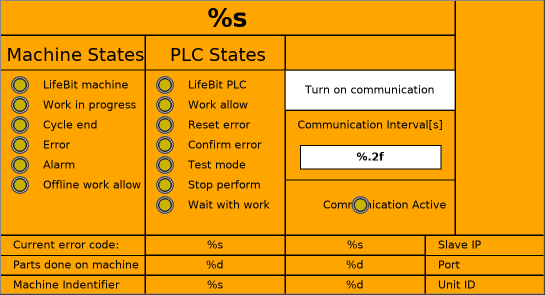
VISUALIZATION vChiniseMachineStatus_v2  // 545x295
VAR_IN_OUT
	stData					:	stChiniseMachineHmiData;
	stParams				:	stModTcpSlaveParams;
END_VAR
    Rectangle (285,35 170x200)
    Rectangle (0,235 145x60)
    Rectangle (0,35 145x200)
    Rectangle (0,35 455x35)
    Rectangle (145,35 140x200)
    Lamp1 (10,75 20x20), variable: stData.stPimCommunicationData.bLifeBitMachine, style: Lamp-Lamp1-Yellow
    Label (40,75 150x20), "LifeBit machine"
    Label (5,40 141x30), "Machine States"
    Lamp1 (10,95 20x20), variable: stData.stPimCommunicationData.bWorkInProgress, style: Lamp-Lamp1-Yellow
    Label (40,95 150x20), "Work in progress"
    Lamp1 (10,115 20x20), variable: stData.stPimCommunicationData.bCycleEnd, style: Lamp-Lamp1-Yellow
    Label (40,115 150x20), "Cycle end"
    Lamp1 (10,135 20x20), variable: stData.stPimCommunicationData.bError, style: Lamp-Lamp1-Yellow
    Label (40,135 150x20), "Error"
    Lamp1 (10,155 20x20), variable: stData.stPimCommunicationData.bAlarm, style: Lamp-Lamp1-Yellow
    Label (40,155 150x20), "Alarm"
    Lamp1 (10,175 20x20), variable: stData.stPimCommunicationData.bOfflineWorkAllow, style: Lamp-Lamp1-Yellow
    Label (40,175 150x20), "Offline work allow"
    Lamp1 (155,75 20x20), variable: stData.stPimCommunicationData.bLifeBitPLC, style: Lamp-Lamp1-Yellow
    Label (185,75 150x20), "LifeBit PLC"
    Label (150,40 136x30), "PLC States"
    Lamp1 (155,95 20x20), variable: stData.stPimCommunicationData.bWorkAllow, style: Lamp-Lamp1-Yellow
    Label (185,95 150x20), "Work allow"
    Lamp1 (155,115 20x20), variable: stData.stPimCommunicationData.bResetError, style: Lamp-Lamp1-Yellow
    Label (185,115 150x20), "Reset error"
    Lamp1 (155,135 20x20), variable: stData.stPimCommunicationData.bConfirmError, style: Lamp-Lamp1-Yellow
    Label (185,135 150x20), "Confirm error"
    Lamp1 (155,155 20x20), variable: stData.stPimCommunicationData.bTestMode, style: Lamp-Lamp1-Yellow
    Label (185,155 150x20), "Test mode"
    Lamp1 (155,175 20x20), variable: stData.stPimCommunicationData.bStopPerform, style: Lamp-Lamp1-Yellow
    Label (185,175 150x20), "Stop perform"
    Lamp1 (155,195 20x20), variable: stData.stPimCommunicationData.bWaitWithWork, style: Lamp-Lamp1-Yellow
    Label (185,195 150x20), "Wait with work"
    Rectangle (145,235 140x20), "%s", text variable: stData.stPimCommunicationData.iErrorCode
    Label (10,235 150x20), "Current error code:"
    Rectangle (0,0 455x35), "%s", text variable: stData.stModbusTcpData.sMachineIndifiner
    Rectangle (145,275 140x20), "%s", text variable: stData.stModbusTcpData.sMachineIndifiner
    Rectangle (285,235 140x20), "%s", text variable: stData.stModbusTcpData.sIpAdress
    Rectangle (285,255 140x20), "%d", text variable: stData.stModbusTcpData.iPort
    Rectangle (285,275 140x20), "%d", text variable: stData.stModbusTcpData.iUnitId
    Rectangle (425,235 120x60)
    Label (10,275 150x20), "Machine Indentifier"
    Label (435,235 86x20), "Slave IP"
    Rectangle (285,70 170x40), "Turn on communication"
        OnMouseClick: toggle stParams.bCommunicationActive
    Label (435,275 101x20), "Unit ID"
    Label (435,255 86x20), "Port"
    Label (320,195 141x20), "Communication Active"
    Lamp1 (290,195 141x20), variable: stParams.bCommunicationActive, style: Lamp-Lamp1-Yellow
    Rectangle (285,110 170x70)
    Rectangle (300,145 141x24), "%.2f", text variable: stParams.rCommunicationCycleTime
        OnMouseClick: write the text variable via Default, format %d
    Label (300,115 141x20), "Communication Interval[s]"
    Rectangle (145,255 140x20), "%d", text variable: stData.stPimCommunicationData.wGoodPartsAmount
    Label (10,255 150x20), "Parts done on machine"
    Rectangle (455,0 90x235)
    Rectangle (425,275 120x20)
    Rectangle (425,255 120x20)
    Rectangle (0,275 145x20)
    Rectangle (0,255 145x20)
END_VISUALIZATION

(* stored: Version 1.1.0.1, ProductVersion 3.1.4024.13
   Visu vChiniseMachineStatus_v2: Id {dcf184be-0a67-4b1f-abc2-f7a6bff23822} *)
